PROGRAM prg_ADS
VAR
	ADS_1: FB_ADS_Read;
	str_ADS_read: STRING(40);
	byte_array : ARRAY[0..1023] OF BYTE;
	struct_received	: struct_ADS_Anker;						
	int_liveCount		: INT;						//{#lynus.ag#()}
	byte_old: BYTE;
END_VAR


str_ADS_read := 'prgComEffIO.byte_array';

ADS_1(
	udintWriteLength:=  SIZEOF(byte_array), 
	udintReadLength:= SIZEOF(byte_array), 
	dwSourceAddr:= ADR(str_ADS_read), 
	dwDestAddr:= ADR(byte_array), 
	strNetID:= '5.146.122.188.1.1', // EIOAN010009 Meidlinger Hauptstraße 77-79 Meidlinger Hauptstraße 77-79        Filiale 5261
	timeReadDelay:= T#5S, 
	mADSError=> , 
	strADSErrorText=> );
	
// copy struct to byte array
IF byte_array[1] <> byte_old AND NOT ADS_1.mADSError AND byte_array[1] <> 0 THEN
	IF SIZEOF(struct_received) > SIZEOF(byte_array) THEN
		memcpy(ADR(struct_received),ADR(byte_array),SIZEOF(byte_array));
	ELSE
		memcpy(ADR(struct_received),ADR(byte_array),SIZEOF(struct_received));
	END_IF
	byte_old := byte_array[1];
END_IF
	
	
int_liveCount := prg_ADS.struct_received.int_liveCount 	;

END_PROGRAM

(* stored: Version 1.1.0.1, ProductVersion 3.1.4024.12
   POU prg_ADS: Id {d3dc75c9-47b8-4f35-adf8-9404eded95fc}, SpecialFunc None *)
